TYPE ST_AirPressureHal :
STRUCT
    LowPressure : BOOL;
    OperatingPressure : BOOL;
    Quality : BOOL := TRUE;
END_STRUCT
END_TYPE

(* stored: Version 1.1.0.1, ProductVersion 3.1.4024.12
   DUT ST_AirPressureHal: Id {580274b2-c7d9-42e8-b7bc-5c106834d946} *)
